// TIA Portal V18 export
TYPE "UDT_AHUsDI"
// stored: IsFailsafeCompliant false
   STRUCT
      xHeaterPumpReady : Array[1..3] of Bool;
      xHeaterPumpInd : Array[1..3] of Bool;
      xHeaterPumpAlarm : Array[1..3] of Bool;
      xSAFAnalogReady : Array[1..3] of Bool;
      xSAFAnalogInd : Array[1..3] of Bool;
      xSAFAnalogAlarm : Array[1..3] of Bool;
      xSAFSp1Ready : Array[1..3] of Bool;
      xSAFSp1Ind : Array[1..3] of Bool;
      xSAFSp1Alarm : Array[1..3] of Bool;
      xSAFSp2Ready : Array[1..3] of Bool;
      xSAFSp2Ind : Array[1..3] of Bool;
      xSAFSp2Alarm : Array[1..3] of Bool;
      xSAFdPInd : Array[1..3] of Bool;
      xFrostProtTstat : Array[1..3] of Bool;
      xSAFdPAlarm : Array[1..3] of Bool;
      xSAFPanelSelectorOff : Array[1..3] of Bool;
      xSAFPanelSelector1St : Array[1..3] of Bool;
      xSAFPanelSelector2St : Array[1..3] of Bool;
      xSAFPanelSelectorAuto : Array[1..3] of Bool;
      xSAFMotorPTCAlarm : Array[1..3] of Bool;
      xReserve1 : Array[1..3] of Bool;
   END_STRUCT;
END_TYPE
